PROGRAM P_Demo_FB_DMXSetIdentifyDevice
VAR
    fbSetIdentify     : FB_DMXSetIdentifyDevice;      // 置 / 复位识别
    stDmxCmdBuffer    : ST_DMXCommandBuffer;          // 与通讯 FB 共用
    wTargetManufId    : WORD := 16#4241;              // 目标灯具厂商 ID
    dwTargetDeviceId  : DWORD := 16#12131415;         // 目标灯具设备 ID
    byTargetPort      : BYTE := 0;                    // 根设备通道 0
    bIdentifyOn       : BOOL := TRUE;                 // TRUE=进入识别(闪烁)
    bDoSet            : BOOL := FALSE;                // 在线给一次上升沿触发
    bBusy             : BOOL;
    bError            : BOOL;
    udiErrId          : UDINT;
END_VAR

// ============================================================
// Tc2_DMX.FB_DMXSetIdentifyDevice 演示程序
// ============================================================
// 场景：维护时在几十台灯里找到 PLC 报警指向的那台：对该 UID 发识别(闪烁)，定位完再关。
// 价值：把让某台灯自报家门做成一次 PLC 调用，免去现场逐台拔插或对照地址表。
// 验证：给 bDoSet 一次上升沿（bIdentifyOn=TRUE）-> bBusy 短暂 TRUE -> 回 FALSE 后现场目标灯应开始闪烁；改 bIdentifyOn=FALSE 再触发可关闭闪烁。
// 验证步骤：
//   1. 右键 PLC 项目下 POUs 文件夹 → Add → Existing Item → 选本 .TcPOU 文件
//   2. 引用 Tc2_DMX；同项目里放一个 FB_EL6851CommunicationEx 实例并共用 stDmxCmdBuffer（非 CycleMode）
//   3. 编译 → 登录 → 运行；按上方『验证』行在线给上升沿观察
// ============================================================

fbSetIdentify(
    bStart                     := bDoSet,
    wDestinationManufacturerId := wTargetManufId,
    dwDestinationDeviceId      := dwTargetDeviceId,
    byPortId                   := byTargetPort,
    bIdentify                  := bIdentifyOn,
    dwOptions                  := 0,
    stCommandBuffer            := stDmxCmdBuffer,
    bBusy                      => bBusy,
    bError                     => bError,
    udiErrorId                 => udiErrId
);

END_PROGRAM

(* stored: Version 1.1.0.1, ProductVersion 3.1.4024.5
   POU P_Demo_FB_DMXSetIdentifyDevice: Id {20222167-e42d-589d-b525-a855eb6a256f}, SpecialFunc None *)
